// TIA Portal V15.1 export
// export: Created 2024-05-17T05:38:22.4671284Z, ExportSetting WithDefaults, DisplayName Totally Integrated Automation Portal, DisplayVersion V15.1 Update 5, DisplayName TIA Portal Openness, DisplayVersion V15.1 Update 5, DisplayName SINAMICS Startdrive Advanced, DisplayVersion V15.1, DisplayName G130, G150, S120, S150, SINAMICS MV, S210, DisplayVersion V15.1, DisplayName G110M, G120, G120C, G120D, G120P, DisplayVersion V15.1, DisplayName STEP 7 Professional, DisplayVersion V15.1 Update 5, DisplayName STEP 7 Safety, DisplayVersion V15.1, DisplayName WinCC Professional, DisplayVersion V15.1 Update 5, DisplayName SIMATIC Visualization Architect, DisplayVersion V15.1
DATA_BLOCK "_209230ASD01"   // DB1942
{ S7_Optimized_Access := 'TRUE' }
VERSION : 0.1
// stored: AutoNumber false, DBAccessibleFromOPCUA true, InstanceOfName LGBGateLock-MGB-Maint, InstanceOfType FB
"LGBGateLock-MGB-Maint"
   // VAR_INPUT
   //    I_SafetyGateInput { ExternalAccessible := 'False'; ExternalVisible := 'False'; ExternalWritable := 'False'} : Bool;
   //    I_Q { ExternalAccessible := 'False'; ExternalVisible := 'False'; ExternalWritable := 'False'} : Bool;
   //    I_EnableAlarm { ExternalAccessible := 'False'; ExternalVisible := 'False'; ExternalWritable := 'False'} : Bool;
   //    I_StartPBInd { ExternalAccessible := 'False'; ExternalVisible := 'False'; ExternalWritable := 'False'} : Bool;
   //    I_AlarmResetPBInd { ExternalAccessible := 'False'; ExternalVisible := 'False'; ExternalWritable := 'False'} : Bool;
   //    I_AccessStopReached { ExternalAccessible := 'False'; ExternalVisible := 'False'; ExternalWritable := 'False'} : Bool;
   //    I_CycleStopRequest { ExternalAccessible := 'False'; ExternalVisible := 'False'; ExternalWritable := 'False'} : Bool;
   //    I_CycleStopReached { ExternalAccessible := 'False'; ExternalVisible := 'False'; ExternalWritable := 'False'} : Bool;
   //    I_MaintRequest { ExternalAccessible := 'False'; ExternalVisible := 'False'; ExternalWritable := 'False'} : Bool;
   //    I_MaintReached { ExternalAccessible := 'False'; ExternalVisible := 'False'; ExternalWritable := 'False'} : Bool;
   //    I_SafetyCard_Pass_Out { ExternalAccessible := 'False'; ExternalVisible := 'False'; ExternalWritable := 'False'} : Bool;
   //    I_SafetyCard_ACK_REQ { ExternalAccessible := 'False'; ExternalVisible := 'False'; ExternalWritable := 'False'} : Bool;
   //    I_SafetyCard_ACK_DIAG { ExternalAccessible := 'False'; ExternalVisible := 'False'; ExternalWritable := 'False'} : Byte;
   //    "C_MGB-B" { ExternalAccessible := 'False'; ExternalVisible := 'False'; ExternalWritable := 'False'} : HW_SUBMODULE;
   //    "C_MGB-EmergencySwitchStd" { ExternalAccessible := 'False'; ExternalVisible := 'False'; ExternalWritable := 'False'} : HW_SUBMODULE;
   //    "C_MGB-L" { ExternalAccessible := 'False'; ExternalVisible := 'False'; ExternalWritable := 'False'} : HW_SUBMODULE;
   //    "C_MBG-EnablingSwitchStd" { ExternalAccessible := 'False'; ExternalVisible := 'False'; ExternalWritable := 'False'} : HW_SUBMODULE;
   //    "C_MBG-DIAG" { ExternalAccessible := 'False'; ExternalVisible := 'False'; ExternalWritable := 'False'} : HW_SUBMODULE;
   // END_VAR
   // VAR_OUTPUT
   //    O_StartPB { ExternalAccessible := 'False'; ExternalVisible := 'False'; ExternalWritable := 'False'} : Bool;
   //    O_ResetAlarmPB { ExternalAccessible := 'False'; ExternalVisible := 'False'; ExternalWritable := 'False'} : Bool;
   //    O_StopPB { ExternalAccessible := 'False'; ExternalVisible := 'False'; ExternalWritable := 'False'} : Bool;
   //    O_EnablingSwitchPB { ExternalAccessible := 'False'; ExternalVisible := 'False'; ExternalWritable := 'False'} : Bool;
   //    "O_EnablingSwitch+PB" { ExternalAccessible := 'False'; ExternalVisible := 'False'; ExternalWritable := 'False'} : Bool;
   //    "O_EnablingSwitch-PB" { ExternalAccessible := 'False'; ExternalVisible := 'False'; ExternalWritable := 'False'} : Bool;
   //    O_MaintReq { ExternalAccessible := 'False'; ExternalVisible := 'False'; ExternalWritable := 'False'} : Bool;
   //    O_CycleStopReq { ExternalAccessible := 'False'; ExternalVisible := 'False'; ExternalWritable := 'False'} : Bool;
   //    O_AccesStopReq { ExternalAccessible := 'False'; ExternalVisible := 'False'; ExternalWritable := 'False'} : Bool;
   //    O_SafetyGateAlarm { ExternalAccessible := 'False'; ExternalVisible := 'False'; ExternalWritable := 'False'} : Bool;
   //    O_EnablingSwitchAlarm { ExternalAccessible := 'False'; ExternalVisible := 'False'; ExternalWritable := 'False'} : Bool;
   //    O_SolenoidAlarm { ExternalAccessible := 'False'; ExternalVisible := 'False'; ExternalWritable := 'False'} : Bool;
   //    O_AccessReqAlarm { ExternalAccessible := 'False'; ExternalVisible := 'False'; ExternalWritable := 'False'} : Bool;
   //    O_MGBDiagWarning { ExternalAccessible := 'False'; ExternalVisible := 'False'; ExternalWritable := 'False'} : Bool;
   //    O_AlarmABCondition { ExternalAccessible := 'False'; ExternalVisible := 'False'; ExternalWritable := 'False'} : Bool;
   // END_VAR
   // VAR_IN_OUT
   //    IO_Modes : "Modes";
   //    H_HMI : "H_HMI";
   //    "H_GateLock-MGB" : "H_GateLock-MGB-Maint";
   //    C_AlarmHighSeverityA { ExternalAccessible := 'False'; ExternalVisible := 'False'; ExternalWritable := 'False'} : Bool;
   //    C_AlarmHighSeverityB { ExternalAccessible := 'False'; ExternalVisible := 'False'; ExternalWritable := 'False'} : Bool;
   //    C_Warning { ExternalAccessible := 'False'; ExternalVisible := 'False'; ExternalWritable := 'False'} : Bool;
   // END_VAR
   // VAR
   //    MGB { ExternalAccessible := 'False'; ExternalVisible := 'False'; ExternalWritable := 'False'} : "Euchner-MGB-Maint";
   //    SafetyCard { ExternalAccessible := 'False'; ExternalVisible := 'False'; ExternalWritable := 'False'} : "SafetyCard";
   //    Pass_Out { ExternalAccessible := 'False'; ExternalVisible := 'False'; ExternalWritable := 'False'} : Bool;
   //    Ack_Req { ExternalAccessible := 'False'; ExternalVisible := 'False'; ExternalWritable := 'False'} : Bool;
   //    Timeout_F_I_O { ExternalAccessible := 'False'; ExternalVisible := 'False'; ExternalWritable := 'False'} : Bool;
   //    ChannelFault_F_I_O { ExternalAccessible := 'False'; ExternalVisible := 'False'; ExternalWritable := 'False'} : Bool;
   //    CRCSeqError_F_I_O { ExternalAccessible := 'False'; ExternalVisible := 'False'; ExternalWritable := 'False'} : Bool;
   //    Timeout_F_Sys { ExternalAccessible := 'False'; ExternalVisible := 'False'; ExternalWritable := 'False'} : Bool;
   //    SeqError_F_Sys { ExternalAccessible := 'False'; ExternalVisible := 'False'; ExternalWritable := 'False'} : Bool;
   //    CRCError_F_Sys { ExternalAccessible := 'False'; ExternalVisible := 'False'; ExternalWritable := 'False'} : Bool;
   //    DelayStop { ExternalAccessible := 'False'; ExternalVisible := 'False'; ExternalWritable := 'False'} : Bool;
   //    DelayMaint { ExternalAccessible := 'False'; ExternalVisible := 'False'; ExternalWritable := 'False'} : Bool;
   //    SafetyGateAlarm { ExternalAccessible := 'False'; ExternalVisible := 'False'; ExternalWritable := 'False'} : Bool;
   //    SafetyGateAlarmCond { ExternalAccessible := 'False'; ExternalVisible := 'False'; ExternalWritable := 'False'} : Bool;
   //    EnablingSwitchAlarm { ExternalAccessible := 'False'; ExternalVisible := 'False'; ExternalWritable := 'False'} : Bool;
   //    EnablingSwitchAlarmCond { ExternalAccessible := 'False'; ExternalVisible := 'False'; ExternalWritable := 'False'} : Bool;
   //    SolenoidAlarm { ExternalAccessible := 'False'; ExternalVisible := 'False'; ExternalWritable := 'False'} : Bool;
   //    SolenoidAlarmCond { ExternalAccessible := 'False'; ExternalVisible := 'False'; ExternalWritable := 'False'} : Bool;
   //    AccessReqAlarm { ExternalAccessible := 'False'; ExternalVisible := 'False'; ExternalWritable := 'False'} : Bool;
   //    DelayCheckGuardUnlocking { ExternalAccessible := 'False'; ExternalVisible := 'False'; ExternalWritable := 'False'} : Bool;
   //    AccessReqSel { ExternalAccessible := 'False'; ExternalVisible := 'False'; ExternalWritable := 'False'} : Bool;
   //    AccessReq { ExternalAccessible := 'False'; ExternalVisible := 'False'; ExternalWritable := 'False'} : Bool;
   //    NotAutoMem { ExternalAccessible := 'False'; ExternalVisible := 'False'; ExternalWritable := 'False'} : Bool;
   //    DelayTimerPbStop { ExternalAccessible := 'False'; ExternalVisible := 'False'; ExternalWritable := 'False'} : IEC_TIMER;
   //    DelayTimerSolenoidAlarm { ExternalAccessible := 'False'; ExternalVisible := 'False'; ExternalWritable := 'False'} : IEC_TIMER;
   //    DelayTimerMaintPb { ExternalAccessible := 'False'; ExternalVisible := 'False'; ExternalWritable := 'False'} : IEC_TIMER;
   //    DelayOFFAutoMode { ExternalAccessible := 'False'; ExternalVisible := 'False'; ExternalWritable := 'False'} : IEC_TIMER;
   //    Edge { ExternalAccessible := 'False'; ExternalVisible := 'False'; ExternalWritable := 'False'} : Array[1..10] of Bool;
   //    _ToggleReqAccess { ExternalAccessible := 'False'; ExternalVisible := 'False'; ExternalWritable := 'False'} : "LToggle";
   // END_VAR
BEGIN
END_DATA_BLOCK
